(* Logix 5000 project; controller PRG_PRESENT Emulate 5570 rev 30.12; software revision 30.00 *)

TASK MainTask (periodic, rate 5000 ms, priority 10, watchdog 5000 ms) : MainProgram

MODULES
   Local : Emulate 5570 (ICP 3, rev 30.12)
       : vendor 1 type 0 code 15 (ICP 0, rev 1.1, Output RPI 50 ms)
END_MODULES

PROGRAM MainProgram   (* main routine MainRoutine *)
VAR
   PRG_Counter : DINT[2];
   PRG_i : DINT;
   PRG_j : DINT;
   PRG_Res_Len : DINT;
   PRG_Result : DINT[128];
   PT_Ciphertext : DINT[2] := ([0] := 1104402914, [1] := 1719681869);
   PT_Enc_i : DINT := 1;
   PT_i : DINT := 32;
   PT_j : DINT := 32;
   PT_Key : DINT[4];
   PT_Key_tmp : DINT[4];
   PT_Pbox : DINT[64] := ([1] := 16, [2] := 32, [3] := 48, [4] := 1, [5] := 17, [6] := 33, [7] := 49, [8] := 2, [9] := 18, [10] := 34, [11] := 50, [12] := 3, [13] := 19, [14] := 35, [15] := 51, [16] := 4, [17] := 20, [18] := 36, [19] := 52, [20] := 5, [21] := 21, [22] := 37, [23] := 53, [24] := 6, [25] := 22, [26] := 38, [27] := 54, [28] := 7, [29] := 23, [30] := 39, [31] := 55, [32] := 8, [33] := 24, [34] := 40, [35] := 56, [36] := 9, [37] := 25, [38] := 41, [39] := 57, [40] := 10, [41] := 26, [42] := 42, [43] := 58, [44] := 11, [45] := 27, [46] := 43, [47] := 59, [48] := 12, [49] := 28, [50] := 44, [51] := 60, [52] := 13, [53] := 29, [54] := 45, [55] := 61, [56] := 14, [57] := 30, [58] := 46, [59] := 62, [60] := 15,
        [61] := 31, [62] := 47, [63] := 63);
   PT_Plaintext : DINT[2] := ([0] := 655340, [1] := -1);
   PT_PState : DINT[2] := ([0] := -1210336382, [1] := 281078171);
   PT_PState_tmp0 : DINT;
   PT_PState_tmp1 : DINT;
   PT_PState_tmp10 : DINT;
   PT_PState_tmp11 : DINT;
   PT_PState_tmp12 : DINT;
   PT_PState_tmp13 : DINT;
   PT_PState_tmp14 : DINT;
   PT_PState_tmp15 : DINT;
   PT_PState_tmp2 : DINT;
   PT_PState_tmp3 : DINT;
   PT_PState_tmp4 : DINT;
   PT_PState_tmp5 : DINT;
   PT_PState_tmp6 : DINT;
   PT_PState_tmp7 : DINT;
   PT_PState_tmp8 : DINT;
   PT_PState_tmp9 : DINT;
   PT_Rd_Key : DINT[2] := ([1] := 452619196);
   PT_Rd_Keys1 : DINT[33,2];
   PT_Rd_Max : DINT := 32;
   PT_round_cnt : DINT;
   PT_Round_Keys : DINT[33,2];
   PT_Sbox : DINT[16] := ([0] := 12, [1] := 5, [2] := 6, [3] := 11, [4] := 9, [6] := 10, [7] := 13, [8] := 3, [9] := 14, [10] := 15, [11] := 8, [12] := 4, [13] := 7, [14] := 1, [15] := 2);
   PT_Sbox_inv : DINT[16] := ([0] := 5, [1] := 14, [2] := 15, [3] := 8, [4] := 12, [5] := 1, [6] := 2, [7] := 13, [8] := 11, [9] := 4, [10] := 6, [11] := 3, [13] := 7, [14] := 9, [15] := 10);
   PT_State : DINT[2] := ([0] := 655340, [1] := -1);
   PT_State_tmp : DINT := 14;
   SCAN_CYCLE_TIME : DINT := 1227;
END_VAR

ROUTINE MainRoutine   (* ladder *)
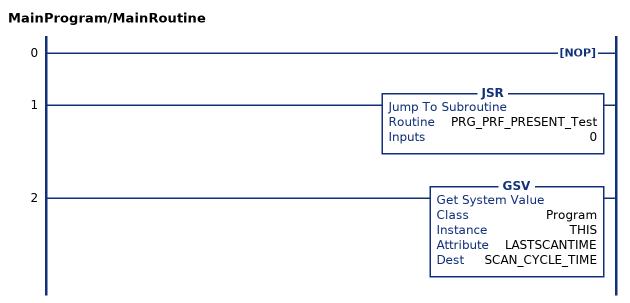
   0: NOP();
   1: JSR(PRG_PRF_PRESENT_Test,0);
   2: GSV(Program,THIS,LASTSCANTIME,SCAN_CYCLE_TIME);
END_ROUTINE

ROUTINE PRESENT_AddRoundKey   (* structured text *)
   
   
   PT_State[0]:=PT_State[0] XOR PT_Rd_Key[0];
   
   
   PT_State[1]:=PT_State[1] XOR PT_Rd_Key[1];
   
END_ROUTINE

ROUTINE PRESENT_ClearKey   (* structured text *)
   PT_Rd_Key[0]:=0;      // round key
   PT_Rd_Key[0]:=0;
END_ROUTINE

ROUTINE PRESENT_Enc   (* structured text *)
   //JSR(Present_Init);        //Init params
   
   PT_State[0]:=PT_Plaintext[0];
   PT_State[1]:=PT_Plaintext[1];
   
   For PT_Enc_i:=1 to PT_Rd_Max-1 by 1 do
   	JSR(PRESENT_GetRoundKey);
   	JSR(PRESENT_AddRoundKey);
   	JSR(PRESENT_SPLayer);
   	PT_Round_Keys[PT_Enc_i,0]:=0;
   	PT_Round_Keys[PT_Enc_i,1]:=0;
   End_For;
   
   JSR(PRESENT_GetRoundKey);
   JSR(PRESENT_AddRoundKey);
   PT_Ciphertext[0]:=PT_State[0];
   PT_Ciphertext[1]:=PT_State[1];
   
   PT_Round_Keys[PT_Enc_i,0]:=0;
   PT_Round_Keys[PT_Enc_i,1]:=0;
   
   
   
   JSR(PRESENT_ClearKey);
   
   
   
   
   
   
END_ROUTINE

ROUTINE PRESENT_GetRoundKey   (* structured text *)
   PT_Rd_Key[0]:=PT_Round_Keys[PT_Enc_i,0];
   PT_Rd_Key[1]:=PT_Round_Keys[PT_Enc_i,1];
   
   PT_Round_Keys[PT_Enc_i,0]:=0;
   PT_Round_Keys[PT_Enc_i,1]:=0;
END_ROUTINE

ROUTINE PRESENT_Init   (* structured text *)
   PT_Sbox[0]:=12;
   PT_Sbox[1]:=5;
   PT_Sbox[2]:=6;
   PT_Sbox[3]:=11;
   PT_Sbox[4]:=9;
   PT_Sbox[5]:=0;
   PT_Sbox[6]:=10;
   PT_Sbox[7]:=13;
   PT_Sbox[8]:=3;
   PT_Sbox[9]:=14;
   PT_Sbox[10]:=15;
   PT_Sbox[11]:=8;
   PT_Sbox[12]:=4;
   PT_Sbox[13]:=7;
   PT_Sbox[14]:=1;
   PT_Sbox[15]:=2;
   PT_Sbox_inv[0]:=5;
   PT_Sbox_inv[1]:=14;
   PT_Sbox_inv[2]:=15;
   PT_Sbox_inv[3]:=8;
   PT_Sbox_inv[4]:=12;
   PT_Sbox_inv[5]:=1;
   PT_Sbox_inv[6]:=2;
   PT_Sbox_inv[7]:=13;
   PT_Sbox_inv[8]:=11;
   PT_Sbox_inv[9]:=4;
   PT_Sbox_inv[10]:=6;
   PT_Sbox_inv[11]:=3;
   PT_Sbox_inv[12]:=0;
   PT_Sbox_inv[13]:=7;
   PT_Sbox_inv[14]:=9;
   PT_Sbox_inv[15]:=10;
   PT_Round_Keys[1,0]:=1611756040;
   PT_Round_Keys[1,1]:=-809488967;
   PT_Round_Keys[2,0]:=1114144300;
   PT_Round_Keys[2,1]:=-901940416;
   PT_Round_Keys[3,0]:=1350188135;
   PT_Round_Keys[3,1]:=-1766580660;
   PT_Round_Keys[4,0]:=-2015015113;
   PT_Round_Keys[4,1]:=-791572170;
   PT_Round_Keys[5,0]:=-547957295;
   PT_Round_Keys[5,1]:=1319780843;
   PT_Round_Keys[6,0]:=1483745500;
   PT_Round_Keys[6,1]:=-1850130972;
   PT_Round_Keys[7,0]:=584609113;
   PT_Round_Keys[7,1]:=-888964175;
   PT_Round_Keys[8,0]:=-1271248392;
   PT_Round_Keys[8,1]:=-739763638;
   PT_Round_Keys[9,0]:=-1137890669;
   PT_Round_Keys[9,1]:=-361507197;
   PT_Round_Keys[10,0]:=2062302844;
   PT_Round_Keys[10,1]:=1952827266;
   PT_Round_Keys[11,0]:=-2104974389;
   PT_Round_Keys[11,1]:=1558552730;
   PT_Round_Keys[12,0]:=-861495324;
   PT_Round_Keys[12,1]:=71414296;
   PT_Round_Keys[13,0]:=592307794;
   PT_Round_Keys[13,1]:=-185782097;
   PT_Round_Keys[14,0]:=584128754;
   PT_Round_Keys[14,1]:=-534363177;
   PT_Round_Keys[15,0]:=-2044357525;
   PT_Round_Keys[15,1]:=-663069210;
   PT_Round_Keys[16,0]:=-1545986668;
   PT_Round_Keys[16,1]:=-246696470;
   PT_Round_Keys[17,0]:=1527332130;
   PT_Round_Keys[17,1]:=2039731156;
   PT_Round_Keys[18,0]:=-415528690;
   PT_Round_Keys[18,1]:=288528924;
   PT_Round_Keys[19,0]:=-1870767607;
   PT_Round_Keys[19,1]:=-1442449288;
   PT_Round_Keys[20,0]:=833314432;
   PT_Round_Keys[20,1]:=1809800897;
   PT_Round_Keys[21,0]:=441101910;
   PT_Round_Keys[21,1]:=900623816;
   PT_Round_Keys[22,0]:=-790238630;
   PT_Round_Keys[22,1]:=-1189262734;
   PT_Round_Keys[23,0]:=-242508722;
   PT_Round_Keys[23,1]:=1139766780;
   PT_Round_Keys[24,0]:=-812600157;
   PT_Round_Keys[24,1]:=-231420497;
   PT_Round_Keys[25,0]:=-1228657155;
   PT_Round_Keys[25,1]:=633425907;
   PT_Round_Keys[26,0]:=1761719627;
   PT_Round_Keys[26,1]:=1984967746;
   PT_Round_Keys[27,0]:=-1201161406;
   PT_Round_Keys[27,1]:=374667251;
   PT_Round_Keys[28,0]:=-2021531509;
   PT_Round_Keys[28,1]:=-119833869;
   PT_Round_Keys[29,0]:=-1564408762;
   PT_Round_Keys[29,1]:=1302627134;
   PT_Round_Keys[30,0]:=-1367541034;
   PT_Round_Keys[30,1]:=1698867279;
   PT_Round_Keys[31,0]:=794755800;
   PT_Round_Keys[31,1]:=-1333752603;
   PT_Round_Keys[32,0]:=1425672852;
   PT_Round_Keys[32,1]:=1740848445;
   
END_ROUTINE

ROUTINE PRESENT_SPLayer   (* structured text *)
   PT_State_tmp.[0]:=PT_State[0].[0];
   PT_State_tmp.[1]:=PT_State[0].[1];
   PT_State_tmp.[2]:=PT_State[0].[2];
   PT_State_tmp.[3]:=PT_State[0].[3];
   PT_State_tmp:=PT_Sbox[PT_State_tmp];
   PT_PState[0].[0]:=PT_State_tmp.[0];
   PT_PState[0].[16]:=PT_State_tmp.[1];
   PT_PState[1].[0]:=PT_State_tmp.[2];
   PT_PState[1].[16]:=PT_State_tmp.[3];
   PT_State_tmp.[0]:=PT_State[0].[4];
   PT_State_tmp.[1]:=PT_State[0].[5];
   PT_State_tmp.[2]:=PT_State[0].[6];
   PT_State_tmp.[3]:=PT_State[0].[7];
   PT_State_tmp:=PT_Sbox[PT_State_tmp];
   PT_PState[0].[1]:=PT_State_tmp.[0];
   PT_PState[0].[17]:=PT_State_tmp.[1];
   PT_PState[1].[1]:=PT_State_tmp.[2];
   PT_PState[1].[17]:=PT_State_tmp.[3];
   PT_State_tmp.[0]:=PT_State[0].[8];
   PT_State_tmp.[1]:=PT_State[0].[9];
   PT_State_tmp.[2]:=PT_State[0].[10];
   PT_State_tmp.[3]:=PT_State[0].[11];
   PT_State_tmp:=PT_Sbox[PT_State_tmp];
   PT_PState[0].[2]:=PT_State_tmp.[0];
   PT_PState[0].[18]:=PT_State_tmp.[1];
   PT_PState[1].[2]:=PT_State_tmp.[2];
   PT_PState[1].[18]:=PT_State_tmp.[3];
   PT_State_tmp.[0]:=PT_State[0].[12];
   PT_State_tmp.[1]:=PT_State[0].[13];
   PT_State_tmp.[2]:=PT_State[0].[14];
   PT_State_tmp.[3]:=PT_State[0].[15];
   PT_State_tmp:=PT_Sbox[PT_State_tmp];
   PT_PState[0].[3]:=PT_State_tmp.[0];
   PT_PState[0].[19]:=PT_State_tmp.[1];
   PT_PState[1].[3]:=PT_State_tmp.[2];
   PT_PState[1].[19]:=PT_State_tmp.[3];
   PT_State_tmp.[0]:=PT_State[0].[16];
   PT_State_tmp.[1]:=PT_State[0].[17];
   PT_State_tmp.[2]:=PT_State[0].[18];
   PT_State_tmp.[3]:=PT_State[0].[19];
   PT_State_tmp:=PT_Sbox[PT_State_tmp];
   PT_PState[0].[4]:=PT_State_tmp.[0];
   PT_PState[0].[20]:=PT_State_tmp.[1];
   PT_PState[1].[4]:=PT_State_tmp.[2];
   PT_PState[1].[20]:=PT_State_tmp.[3];
   PT_State_tmp.[0]:=PT_State[0].[20];
   PT_State_tmp.[1]:=PT_State[0].[21];
   PT_State_tmp.[2]:=PT_State[0].[22];
   PT_State_tmp.[3]:=PT_State[0].[23];
   PT_State_tmp:=PT_Sbox[PT_State_tmp];
   PT_PState[0].[5]:=PT_State_tmp.[0];
   PT_PState[0].[21]:=PT_State_tmp.[1];
   PT_PState[1].[5]:=PT_State_tmp.[2];
   PT_PState[1].[21]:=PT_State_tmp.[3];
   PT_State_tmp.[0]:=PT_State[0].[24];
   PT_State_tmp.[1]:=PT_State[0].[25];
   PT_State_tmp.[2]:=PT_State[0].[26];
   PT_State_tmp.[3]:=PT_State[0].[27];
   PT_State_tmp:=PT_Sbox[PT_State_tmp];
   PT_PState[0].[6]:=PT_State_tmp.[0];
   PT_PState[0].[22]:=PT_State_tmp.[1];
   PT_PState[1].[6]:=PT_State_tmp.[2];
   PT_PState[1].[22]:=PT_State_tmp.[3];
   PT_State_tmp.[0]:=PT_State[0].[28];
   PT_State_tmp.[1]:=PT_State[0].[29];
   PT_State_tmp.[2]:=PT_State[0].[30];
   PT_State_tmp.[3]:=PT_State[0].[31];
   PT_State_tmp:=PT_Sbox[PT_State_tmp];
   PT_PState[0].[7]:=PT_State_tmp.[0];
   PT_PState[0].[23]:=PT_State_tmp.[1];
   PT_PState[1].[7]:=PT_State_tmp.[2];
   PT_PState[1].[23]:=PT_State_tmp.[3];
   PT_State_tmp.[0]:=PT_State[1].[0];
   PT_State_tmp.[1]:=PT_State[1].[1];
   PT_State_tmp.[2]:=PT_State[1].[2];
   PT_State_tmp.[3]:=PT_State[1].[3];
   PT_State_tmp:=PT_Sbox[PT_State_tmp];
   PT_PState[0].[8]:=PT_State_tmp.[0];
   PT_PState[0].[24]:=PT_State_tmp.[1];
   PT_PState[1].[8]:=PT_State_tmp.[2];
   PT_PState[1].[24]:=PT_State_tmp.[3];
   PT_State_tmp.[0]:=PT_State[1].[4];
   PT_State_tmp.[1]:=PT_State[1].[5];
   PT_State_tmp.[2]:=PT_State[1].[6];
   PT_State_tmp.[3]:=PT_State[1].[7];
   PT_State_tmp:=PT_Sbox[PT_State_tmp];
   PT_PState[0].[9]:=PT_State_tmp.[0];
   PT_PState[0].[25]:=PT_State_tmp.[1];
   PT_PState[1].[9]:=PT_State_tmp.[2];
   PT_PState[1].[25]:=PT_State_tmp.[3];
   PT_State_tmp.[0]:=PT_State[1].[8];
   PT_State_tmp.[1]:=PT_State[1].[9];
   PT_State_tmp.[2]:=PT_State[1].[10];
   PT_State_tmp.[3]:=PT_State[1].[11];
   PT_State_tmp:=PT_Sbox[PT_State_tmp];
   PT_PState[0].[10]:=PT_State_tmp.[0];
   PT_PState[0].[26]:=PT_State_tmp.[1];
   PT_PState[1].[10]:=PT_State_tmp.[2];
   PT_PState[1].[26]:=PT_State_tmp.[3];
   PT_State_tmp.[0]:=PT_State[1].[12];
   PT_State_tmp.[1]:=PT_State[1].[13];
   PT_State_tmp.[2]:=PT_State[1].[14];
   PT_State_tmp.[3]:=PT_State[1].[15];
   PT_State_tmp:=PT_Sbox[PT_State_tmp];
   PT_PState[0].[11]:=PT_State_tmp.[0];
   PT_PState[0].[27]:=PT_State_tmp.[1];
   PT_PState[1].[11]:=PT_State_tmp.[2];
   PT_PState[1].[27]:=PT_State_tmp.[3];
   PT_State_tmp.[0]:=PT_State[1].[16];
   PT_State_tmp.[1]:=PT_State[1].[17];
   PT_State_tmp.[2]:=PT_State[1].[18];
   PT_State_tmp.[3]:=PT_State[1].[19];
   PT_State_tmp:=PT_Sbox[PT_State_tmp];
   PT_PState[0].[12]:=PT_State_tmp.[0];
   PT_PState[0].[28]:=PT_State_tmp.[1];
   PT_PState[1].[12]:=PT_State_tmp.[2];
   PT_PState[1].[28]:=PT_State_tmp.[3];
   PT_State_tmp.[0]:=PT_State[1].[20];
   PT_State_tmp.[1]:=PT_State[1].[21];
   PT_State_tmp.[2]:=PT_State[1].[22];
   PT_State_tmp.[3]:=PT_State[1].[23];
   PT_State_tmp:=PT_Sbox[PT_State_tmp];
   PT_PState[0].[13]:=PT_State_tmp.[0];
   PT_PState[0].[29]:=PT_State_tmp.[1];
   PT_PState[1].[13]:=PT_State_tmp.[2];
   PT_PState[1].[29]:=PT_State_tmp.[3];
   PT_State_tmp.[0]:=PT_State[1].[24];
   PT_State_tmp.[1]:=PT_State[1].[25];
   PT_State_tmp.[2]:=PT_State[1].[26];
   PT_State_tmp.[3]:=PT_State[1].[27];
   PT_State_tmp:=PT_Sbox[PT_State_tmp];
   PT_PState[0].[14]:=PT_State_tmp.[0];
   PT_PState[0].[30]:=PT_State_tmp.[1];
   PT_PState[1].[14]:=PT_State_tmp.[2];
   PT_PState[1].[30]:=PT_State_tmp.[3];
   PT_State_tmp.[0]:=PT_State[1].[28];
   PT_State_tmp.[1]:=PT_State[1].[29];
   PT_State_tmp.[2]:=PT_State[1].[30];
   PT_State_tmp.[3]:=PT_State[1].[31];
   PT_State_tmp:=PT_Sbox[PT_State_tmp];
   PT_PState[0].[15]:=PT_State_tmp.[0];
   PT_PState[0].[31]:=PT_State_tmp.[1];
   PT_PState[1].[15]:=PT_State_tmp.[2];
   PT_PState[1].[31]:=PT_State_tmp.[3];
   PT_State[0]:=PT_PState[0];
   PT_State[1]:=PT_PState[1];
   
END_ROUTINE

ROUTINE PRESENT_SPLayer_Inv   (* structured text *)
   PT_PState_tmp0.[0]:=PT_State[0].[0];
   PT_PState_tmp1.[0]:=PT_State[0].[1];
   PT_PState_tmp2.[0]:=PT_State[0].[2];
   PT_PState_tmp3.[0]:=PT_State[0].[3];
   PT_PState_tmp4.[0]:=PT_State[0].[4];
   PT_PState_tmp5.[0]:=PT_State[0].[5];
   PT_PState_tmp6.[0]:=PT_State[0].[6];
   PT_PState_tmp7.[0]:=PT_State[0].[7];
   PT_PState_tmp8.[0]:=PT_State[0].[8];
   PT_PState_tmp9.[0]:=PT_State[0].[9];
   PT_PState_tmp10.[0]:=PT_State[0].[10];
   PT_PState_tmp11.[0]:=PT_State[0].[11];
   PT_PState_tmp12.[0]:=PT_State[0].[12];
   PT_PState_tmp13.[0]:=PT_State[0].[13];
   PT_PState_tmp14.[0]:=PT_State[0].[14];
   PT_PState_tmp15.[0]:=PT_State[0].[15];
   PT_PState_tmp0.[1]:=PT_State[0].[16];
   PT_PState_tmp1.[1]:=PT_State[0].[17];
   PT_PState_tmp2.[1]:=PT_State[0].[18];
   PT_PState_tmp3.[1]:=PT_State[0].[19];
   PT_PState_tmp4.[1]:=PT_State[0].[20];
   PT_PState_tmp5.[1]:=PT_State[0].[21];
   PT_PState_tmp6.[1]:=PT_State[0].[22];
   PT_PState_tmp7.[1]:=PT_State[0].[23];
   PT_PState_tmp8.[1]:=PT_State[0].[24];
   PT_PState_tmp9.[1]:=PT_State[0].[25];
   PT_PState_tmp10.[1]:=PT_State[0].[26];
   PT_PState_tmp11.[1]:=PT_State[0].[27];
   PT_PState_tmp12.[1]:=PT_State[0].[28];
   PT_PState_tmp13.[1]:=PT_State[0].[29];
   PT_PState_tmp14.[1]:=PT_State[0].[30];
   PT_PState_tmp15.[1]:=PT_State[0].[31];
   PT_PState_tmp0.[2]:=PT_State[1].[0];
   PT_PState_tmp1.[2]:=PT_State[1].[1];
   PT_PState_tmp2.[2]:=PT_State[1].[2];
   PT_PState_tmp3.[2]:=PT_State[1].[3];
   PT_PState_tmp4.[2]:=PT_State[1].[4];
   PT_PState_tmp5.[2]:=PT_State[1].[5];
   PT_PState_tmp6.[2]:=PT_State[1].[6];
   PT_PState_tmp7.[2]:=PT_State[1].[7];
   PT_PState_tmp8.[2]:=PT_State[1].[8];
   PT_PState_tmp9.[2]:=PT_State[1].[9];
   PT_PState_tmp10.[2]:=PT_State[1].[10];
   PT_PState_tmp11.[2]:=PT_State[1].[11];
   PT_PState_tmp12.[2]:=PT_State[1].[12];
   PT_PState_tmp13.[2]:=PT_State[1].[13];
   PT_PState_tmp14.[2]:=PT_State[1].[14];
   PT_PState_tmp15.[2]:=PT_State[1].[15];
   PT_PState_tmp0.[3]:=PT_State[1].[16];
   PT_PState_tmp1.[3]:=PT_State[1].[17];
   PT_PState_tmp2.[3]:=PT_State[1].[18];
   PT_PState_tmp3.[3]:=PT_State[1].[19];
   PT_PState_tmp4.[3]:=PT_State[1].[20];
   PT_PState_tmp5.[3]:=PT_State[1].[21];
   PT_PState_tmp6.[3]:=PT_State[1].[22];
   PT_PState_tmp7.[3]:=PT_State[1].[23];
   PT_PState_tmp8.[3]:=PT_State[1].[24];
   PT_PState_tmp9.[3]:=PT_State[1].[25];
   PT_PState_tmp10.[3]:=PT_State[1].[26];
   PT_PState_tmp11.[3]:=PT_State[1].[27];
   PT_PState_tmp12.[3]:=PT_State[1].[28];
   PT_PState_tmp13.[3]:=PT_State[1].[29];
   PT_PState_tmp14.[3]:=PT_State[1].[30];
   PT_PState_tmp15.[3]:=PT_State[1].[31];
   PT_State_tmp:=PT_Sbox_inv[PT_PState_tmp0];
   PT_State[0].[0]:=PT_State_tmp.[0];
   PT_State[0].[1]:=PT_State_tmp.[1];
   PT_State[0].[2]:=PT_State_tmp.[2];
   PT_State[0].[3]:=PT_State_tmp.[3];
   PT_State_tmp:=PT_Sbox_inv[PT_PState_tmp1];
   PT_State[0].[4]:=PT_State_tmp.[0];
   PT_State[0].[5]:=PT_State_tmp.[1];
   PT_State[0].[6]:=PT_State_tmp.[2];
   PT_State[0].[7]:=PT_State_tmp.[3];
   PT_State_tmp:=PT_Sbox_inv[PT_PState_tmp2];
   PT_State[0].[8]:=PT_State_tmp.[0];
   PT_State[0].[9]:=PT_State_tmp.[1];
   PT_State[0].[10]:=PT_State_tmp.[2];
   PT_State[0].[11]:=PT_State_tmp.[3];
   PT_State_tmp:=PT_Sbox_inv[PT_PState_tmp3];
   PT_State[0].[12]:=PT_State_tmp.[0];
   PT_State[0].[13]:=PT_State_tmp.[1];
   PT_State[0].[14]:=PT_State_tmp.[2];
   PT_State[0].[15]:=PT_State_tmp.[3];
   PT_State_tmp:=PT_Sbox_inv[PT_PState_tmp4];
   PT_State[0].[16]:=PT_State_tmp.[0];
   PT_State[0].[17]:=PT_State_tmp.[1];
   PT_State[0].[18]:=PT_State_tmp.[2];
   PT_State[0].[19]:=PT_State_tmp.[3];
   PT_State_tmp:=PT_Sbox_inv[PT_PState_tmp5];
   PT_State[0].[20]:=PT_State_tmp.[0];
   PT_State[0].[21]:=PT_State_tmp.[1];
   PT_State[0].[22]:=PT_State_tmp.[2];
   PT_State[0].[23]:=PT_State_tmp.[3];
   PT_State_tmp:=PT_Sbox_inv[PT_PState_tmp6];
   PT_State[0].[24]:=PT_State_tmp.[0];
   PT_State[0].[25]:=PT_State_tmp.[1];
   PT_State[0].[26]:=PT_State_tmp.[2];
   PT_State[0].[27]:=PT_State_tmp.[3];
   PT_State_tmp:=PT_Sbox_inv[PT_PState_tmp7];
   PT_State[0].[28]:=PT_State_tmp.[0];
   PT_State[0].[29]:=PT_State_tmp.[1];
   PT_State[0].[30]:=PT_State_tmp.[2];
   PT_State[0].[31]:=PT_State_tmp.[3];
   PT_State_tmp:=PT_Sbox_inv[PT_PState_tmp8];
   PT_State[1].[0]:=PT_State_tmp.[0];
   PT_State[1].[1]:=PT_State_tmp.[1];
   PT_State[1].[2]:=PT_State_tmp.[2];
   PT_State[1].[3]:=PT_State_tmp.[3];
   PT_State_tmp:=PT_Sbox_inv[PT_PState_tmp9];
   PT_State[1].[4]:=PT_State_tmp.[0];
   PT_State[1].[5]:=PT_State_tmp.[1];
   PT_State[1].[6]:=PT_State_tmp.[2];
   PT_State[1].[7]:=PT_State_tmp.[3];
   PT_State_tmp:=PT_Sbox_inv[PT_PState_tmp10];
   PT_State[1].[8]:=PT_State_tmp.[0];
   PT_State[1].[9]:=PT_State_tmp.[1];
   PT_State[1].[10]:=PT_State_tmp.[2];
   PT_State[1].[11]:=PT_State_tmp.[3];
   PT_State_tmp:=PT_Sbox_inv[PT_PState_tmp11];
   PT_State[1].[12]:=PT_State_tmp.[0];
   PT_State[1].[13]:=PT_State_tmp.[1];
   PT_State[1].[14]:=PT_State_tmp.[2];
   PT_State[1].[15]:=PT_State_tmp.[3];
   PT_State_tmp:=PT_Sbox_inv[PT_PState_tmp12];
   PT_State[1].[16]:=PT_State_tmp.[0];
   PT_State[1].[17]:=PT_State_tmp.[1];
   PT_State[1].[18]:=PT_State_tmp.[2];
   PT_State[1].[19]:=PT_State_tmp.[3];
   PT_State_tmp:=PT_Sbox_inv[PT_PState_tmp13];
   PT_State[1].[20]:=PT_State_tmp.[0];
   PT_State[1].[21]:=PT_State_tmp.[1];
   PT_State[1].[22]:=PT_State_tmp.[2];
   PT_State[1].[23]:=PT_State_tmp.[3];
   PT_State_tmp:=PT_Sbox_inv[PT_PState_tmp14];
   PT_State[1].[24]:=PT_State_tmp.[0];
   PT_State[1].[25]:=PT_State_tmp.[1];
   PT_State[1].[26]:=PT_State_tmp.[2];
   PT_State[1].[27]:=PT_State_tmp.[3];
   PT_State_tmp:=PT_Sbox_inv[PT_PState_tmp15];
   PT_State[1].[28]:=PT_State_tmp.[0];
   PT_State[1].[29]:=PT_State_tmp.[1];
   PT_State[1].[30]:=PT_State_tmp.[2];
   PT_State[1].[31]:=PT_State_tmp.[3];
   
END_ROUTINE

ROUTINE PRG_PRF_Init   (* structured text *)
   // init PRG_Count[0] and PRG_Count[1] during application.. for PRF.. they could be any values
   //For PRG application, PRG_Count[0] defines the output length (i.e., the number of 64-bit, e.g., 128-bit output, PRG_Count[0]:=2)
   
   //initialize version
   
   PRG_j:=0;
   PRG_Res_Len :=  (PRG_Counter[0] AND 16#0000ffff)-1;
   
   JSR(PRESENT_Init);
END_ROUTINE

ROUTINE PRG_PRF_PRESENT   (* structured text *)
   
   JSR(PRG_PRF_Init);
   
   
   For PRG_i:=0 to PRG_Res_Len by 1 do
   
   	PT_Plaintext[0]:=PRG_Counter[0];
   	PT_Plaintext[1]:=PRG_Counter[1];
   
   	JSR(PRESENT_Enc);
   
   	PRG_Result[PRG_j]:=PT_Ciphertext[0];
   	PRG_Result[PRG_j+1]:=PT_Ciphertext[1];
   
   	PRG_j:=PRG_j+2;
   
   End_For;
   
   JSR(PRESENT_ClearKey);
   
END_ROUTINE

ROUTINE PRG_PRF_PRESENT_Test   (* structured text *)
   If S:FS Then
   
   	PRG_Counter[0]:=5;
   	PRG_Counter[1]:=1;
   
   End_if;
   
   
   JSR(PRG_PRF_PRESENT);
   
   
END_ROUTINE
END_PROGRAM
